FUNCTION_BLOCK PUBLIC Motor
VAR_INPUT
END_VAR
VAR_OUTPUT
END_VAR
VAR
	CurrentlyMoving: BOOL;	// we need this because stepSwitches can be 1 and we should not move
	// Current position is currently stored in the Automatic GVLs.
END_VAR

END_FUNCTION_BLOCK

(* stored: Version 1.1.0.1, ProductVersion 3.1.4024.13
   POU Motor: Id {c9894c91-c290-4e55-869d-cafa71223417}, SpecialFunc None *)
